(* This Function block provides basic  control for Scroll Pumps *)
(* Turn on scroll pump if the Turbo Vent Valve is closed. *)
(* Cannot turn off scroll pump if turb is running. delay scroll off 150s.*)  

FUNCTION_BLOCK FB_ScrollPump
VAR_IN_OUT

END_VAR
VAR_OUTPUT
	{attribute 'pytmc' := '
    pv:
	'}
	iq_stPFO	:	ST_RoughPump;
END_VAR
VAR_INPUT
	TurboIsON : BOOL;
	VentValve	: ST_VCC_NO; // type of vent valve might change
END_VAR
VAR
	Tmr_TOF : TOF;
	tTimerDuration : Time:= T#150S;
	//Previous_RunSW : BOOL;
	// Digital Output to be linked
	q_xRunDo AT%Q*	:   BOOL; 
END_VAR

//Turn on scroll pump if the Turbo Vent Valve is closed. So you are not just
// pumping air and accomplishing nothing

// cannot turn off scroll pump if turb is running. delay scroll off 150s.  


Tmr_TOF(IN:=TurboIsON, PT := tTimerDuration);

IF VentValve.xCLS_DO THEN
	iq_stPFO.q_xRunDo := (Tmr_TOF.Q OR iq_stPFO.pv_xRunSW);
ELSE
	iq_stPFO.q_xRunDo := FALSE;
END_IF

iq_stPFO.pv_xRunSW := iq_stPFO.q_xRunDo;



(*soft io Mapping*)
IO();

ACTION IO:
q_xRunDo:= iq_stPFO.q_xRunDo;
END_ACTION

METHOD PUBLIC M_Run : BOOL
VAR_INPUT
	run:bool; // set to true to run, false to stop;
END_VAR

this^.iq_stPFO.pv_xRunSW := run;
END_METHOD

END_FUNCTION_BLOCK

(* stored: Version 1.1.0.1, ProductVersion 3.1.4022.16
   POU FB_ScrollPump: Id {95800034-a8e9-430e-af6e-1fa7a649fe90}, SpecialFunc None
   Action IO: Id {47ae7053-5350-4e8f-94b2-400e5380039f}
   Method M_Run: Id {eba797a4-1012-42f7-b194-fa0d2f89ba57} *)
